(* IEC 61131-3 sources: com.logicals.lc3.webinar/usRTS_RPMControl_iSOC/src_FB_LIB_SAFE/Compare/USINT, 6 files *)

(* ---- wEQ_USINT_2.iecst ---- *)
NAMESPACE logicals.web.standard
NAMESPACE compare

/*
 * Function block wrapper for IEC 61131-3 EQ<br>
 * IN1 =  1st value (USINT)<br>
 * IN2 =  2nd value (USINT)<br>
 * OUT = true if IN1 is equal to IN2 (BOOL)<br>
 */
FUNCTION_BLOCK wEQ_USINT_2
	{ vNameAlignment:="center"; altName:="="; bgColor:="Plum"; width:=40; hideIONames; }
	VAR_INPUT
		IN1 : USINT;
		IN2 : USINT;
	END_VAR
	VAR_OUTPUT
		OUT : BOOL;
	END_VAR

	OUT := EQ(IN1:=IN1, IN2:=IN2, ENO=>ENO);
END_FUNCTION_BLOCK

END_NAMESPACE
END_NAMESPACE

(* ---- wGE_USINT_2.iecst ---- *)
NAMESPACE logicals.web.standard
NAMESPACE compare

/*
 * Function block wrapper for IEC 61131-3 GE<br>
 * IN1 =  1st value (USINT)<br>
 * IN2 =  2nd value (USINT)<br>
 * OUT = true if IN1 >= IN2 (BOOL)<br>
 */
FUNCTION_BLOCK wGE_USINT_2
	{ vNameAlignment:="center"; altName:=">="; bgColor:="Plum"; width:=40; hideIONames; }
	VAR_INPUT
		IN1 : USINT;
		IN2 : USINT;
	END_VAR
	VAR_OUTPUT
		OUT : BOOL;
	END_VAR

	OUT := GE(IN1:=IN1, IN2:=IN2, ENO=>ENO);
END_FUNCTION_BLOCK

END_NAMESPACE
END_NAMESPACE

(* ---- wGT_USINT_2.iecst ---- *)
NAMESPACE logicals.web.standard
NAMESPACE compare

/*
 * Function block wrapper for IEC 61131-3 GT<br>
 * IN1 =  1st value (USINT)<br>
 * IN2 =  2nd value (USINT)<br>
 * OUT = true if IN1 > IN2 (BOOL)<br>
 */
FUNCTION_BLOCK wGT_USINT_2
	{ vNameAlignment:="center"; altName:=">"; bgColor:="Plum"; width:=40; hideIONames; }
	VAR_INPUT
		IN1 : USINT;
		IN2 : USINT;
	END_VAR
	VAR_OUTPUT
		OUT : BOOL;
	END_VAR

	OUT := GT(IN1:=IN1, IN2:=IN2, ENO=>ENO);
END_FUNCTION_BLOCK

END_NAMESPACE
END_NAMESPACE

(* ---- wLE_USINT_2.iecst ---- *)
NAMESPACE logicals.web.standard
NAMESPACE compare

/*
 * Function block wrapper for IEC 61131-3 LE<br>
 * IN1 =  1st value (USINT)<br>
 * IN2 =  2nd value (USINT)<br>
 * OUT = true if IN1 <= IN2 (BOOL)<br>
 */
FUNCTION_BLOCK wLE_USINT_2
	{ vNameAlignment:="center"; altName:="<="; bgColor:="Plum"; width:=40; hideIONames; }
	VAR_INPUT
		IN1 : USINT;
		IN2 : USINT;
	END_VAR
	VAR_OUTPUT
		OUT : BOOL;
	END_VAR

	OUT := LE(IN1:=IN1, IN2:=IN2, ENO=>ENO);
END_FUNCTION_BLOCK

END_NAMESPACE
END_NAMESPACE

(* ---- wLT_USINT_2.iecst ---- *)
NAMESPACE logicals.web.standard
NAMESPACE compare

/*
 * Function block wrapper for IEC 61131-3 LT<br>
 * IN1 =  1st value (USINT)<br>
 * IN2 =  2nd value (USINT)<br>
 * OUT = true if IN1 < IN2 (BOOL)<br>
 */
FUNCTION_BLOCK wLT_USINT_2
	{ vNameAlignment:="center"; altName:="<"; bgColor:="Plum"; width:=40; hideIONames; }
	VAR_INPUT
		IN1 : USINT;
		IN2 : USINT;
	END_VAR
	VAR_OUTPUT
		OUT : BOOL;
	END_VAR

	OUT := LT(IN1:=IN1, IN2:=IN2, ENO=>ENO);
END_FUNCTION_BLOCK

END_NAMESPACE
END_NAMESPACE

(* ---- wNE_USINT.iecst ---- *)
NAMESPACE logicals.web.standard
NAMESPACE compare

/*
 * Function block wrapper for IEC 61131-3 NE<br>
 * IN1 = value 1 (USINT)<br>
 * IN2 = value 2 (USINT)<br>
 * OUT = true if IN1 is not equal to IN2 (BOOL)<br>
 */
FUNCTION_BLOCK wNE_USINT
	{ vNameAlignment:="center"; altName:="<>"; bgColor:="Plum"; width:=40; hideIONames; }
	VAR_INPUT
		IN1 : USINT;
		IN2 : USINT;
	END_VAR
	VAR_OUTPUT
		OUT : BOOL;
	END_VAR

	OUT := NE(IN1:=IN1, IN2:=IN2, ENO=>ENO);
END_FUNCTION_BLOCK

END_NAMESPACE
END_NAMESPACE
